PROGRAM MAIN
VAR
	test : UDINT;
	testbool : BOOL;
END_VAR

test := test + 1;
testbool := true;

END_PROGRAM

(* stored: Version 1.1.0.1, ProductVersion 3.1.4024.9
   POU MAIN: Id {76ac14f2-4a0d-441a-9cc2-7827074a0a0b}, SpecialFunc None *)
